{attribute addProperty BoxType "EP1809-0042-0019"}
{attribute addProperty Id "DI_X01AT %I*ARRAY[0..1] OF DI_X_E4AEF59E429496728842949672950DI_X02AT %I*ARRAY[0..1] OF DI_X_E4AEF59E429496728842949672950DI_X03AT %I*ARRAY[0..1] OF DI_X_E4AEF59E429496728842949672950DI_X04AT %I*ARRAY[0..1] OF DI_X_E4AEF59E429496728842949672950DI_X05AT %I*ARRAY[0..1] OF DI_X_E4AEF59E429496728842949672950DI_X06AT %I*ARRAY[0..1] OF DI_X_E4AEF59E429496728842949672950DI_X07AT %I*ARRAY[0..1] OF DI_X_E4AEF59E429496728842949672950DI_X08AT %I*ARRAY[0..1] OF DI_X_E4AEF59E429496728842949672950WcStateAT %I*WcState_98A4DF7520.250InfoDataAT %I*InfoData_192954DE1620"}
{attribute addProperty CRC "3455117243"}
{attribute addProperty SizeInBites "4294967250"}
{attribute addProperty SizeInBytes "34359738362.25"}
TYPE EP1809_09F99349 :
STRUCT
	{attribute addProperty Name "DI_X01"}
	DI_X01 : ARRAY[0..1] OF DI_X_E4AEF59E;
	{attribute addProperty Name "DI_X02"}
	DI_X02 : ARRAY[0..1] OF DI_X_E4AEF59E;
	{attribute addProperty Name "DI_X03"}
	DI_X03 : ARRAY[0..1] OF DI_X_E4AEF59E;
	{attribute addProperty Name "DI_X04"}
	DI_X04 : ARRAY[0..1] OF DI_X_E4AEF59E;
	{attribute addProperty Name "DI_X05"}
	DI_X05 : ARRAY[0..1] OF DI_X_E4AEF59E;
	{attribute addProperty Name "DI_X06"}
	DI_X06 : ARRAY[0..1] OF DI_X_E4AEF59E;
	{attribute addProperty Name "DI_X07"}
	DI_X07 : ARRAY[0..1] OF DI_X_E4AEF59E;
	{attribute addProperty Name "DI_X08"}
	DI_X08 : ARRAY[0..1] OF DI_X_E4AEF59E;
	{attribute addProperty Name "WcState"}
	WcState : WcState_98A4DF75;
	{attribute addProperty Name "InfoData"}
	InfoData : InfoData_192954DE;
END_STRUCT
END_TYPE

(* stored: Version 1.2.0.0, ProductVersion 3.1.4024.9
   DUT EP1809_09F99349: Id {2ac95b07-0e0d-4607-8b3a-bcc96cf8c658} *)
